{attribute 'c++_compatible'}
INTERFACE I_TcpRcv

METHOD NewData : HRESULT
VAR_INPUT
	nData	: UDINT;
	pData	: PVOID;
END_VAR
END_METHOD

END_INTERFACE

(* stored: Version 1.1.0.1, ProductVersion 3.1.4019.2
   Itf I_TcpRcv: Id {b0df10c2-e7a4-4918-80ef-0e00e172ad94}
   Method NewData: Id {feb9d736-8e26-4640-b8c4-77bf5037c5cd} *)
